(* PLC project Unnamed, Unknown Unnamed 1 *)
(* stored: creationDateTime 2025-11-17T12:43:33, modificationDateTime 2025-11-17T18:21:39 *)

PROGRAM Lab1
  VAR
    btn AT %IX0.0 : BOOL := False;
  END_VAR
  VAR
    AllowedPress : BOOL := False;
    pressed : BOOL := False;
    Ped_wait : BOOL := False;
    Pedestrian : BOOL := False;
  END_VAR
  VAR
    north AT %QX0.0 : BOOL := False;
    south AT %QX0.1 : BOOL := False;
    west AT %QX0.2 : BOOL := False;
    east AT %QX0.3 : BOOL := False;
  END_VAR
  VAR
    state : BOOL := False;
    S0 : BOOL := False;
    S1 : BOOL := False;
    T10 : TIME := T#10s;
    T80 : TIME := T#80s;
    Allowed_timer : BOOL := False;
    Timer_cooldown : BOOL := False;
    FF1 : BOOL := False;
    FF2 : BOOL := False;
    FF_output : BOOL := False;
    TON0 : TON;
    TON1 : TON;
    TP0 : TP;
    TP1 : TP;
    R_TRIG1 : R_TRIG;
    R_TRIG0 : R_TRIG;
    R_TRIG2 : R_TRIG;
    R_TRIG3 : R_TRIG;
    R_TRIG4 : R_TRIG;
    R_TRIG5 : R_TRIG;
  END_VAR

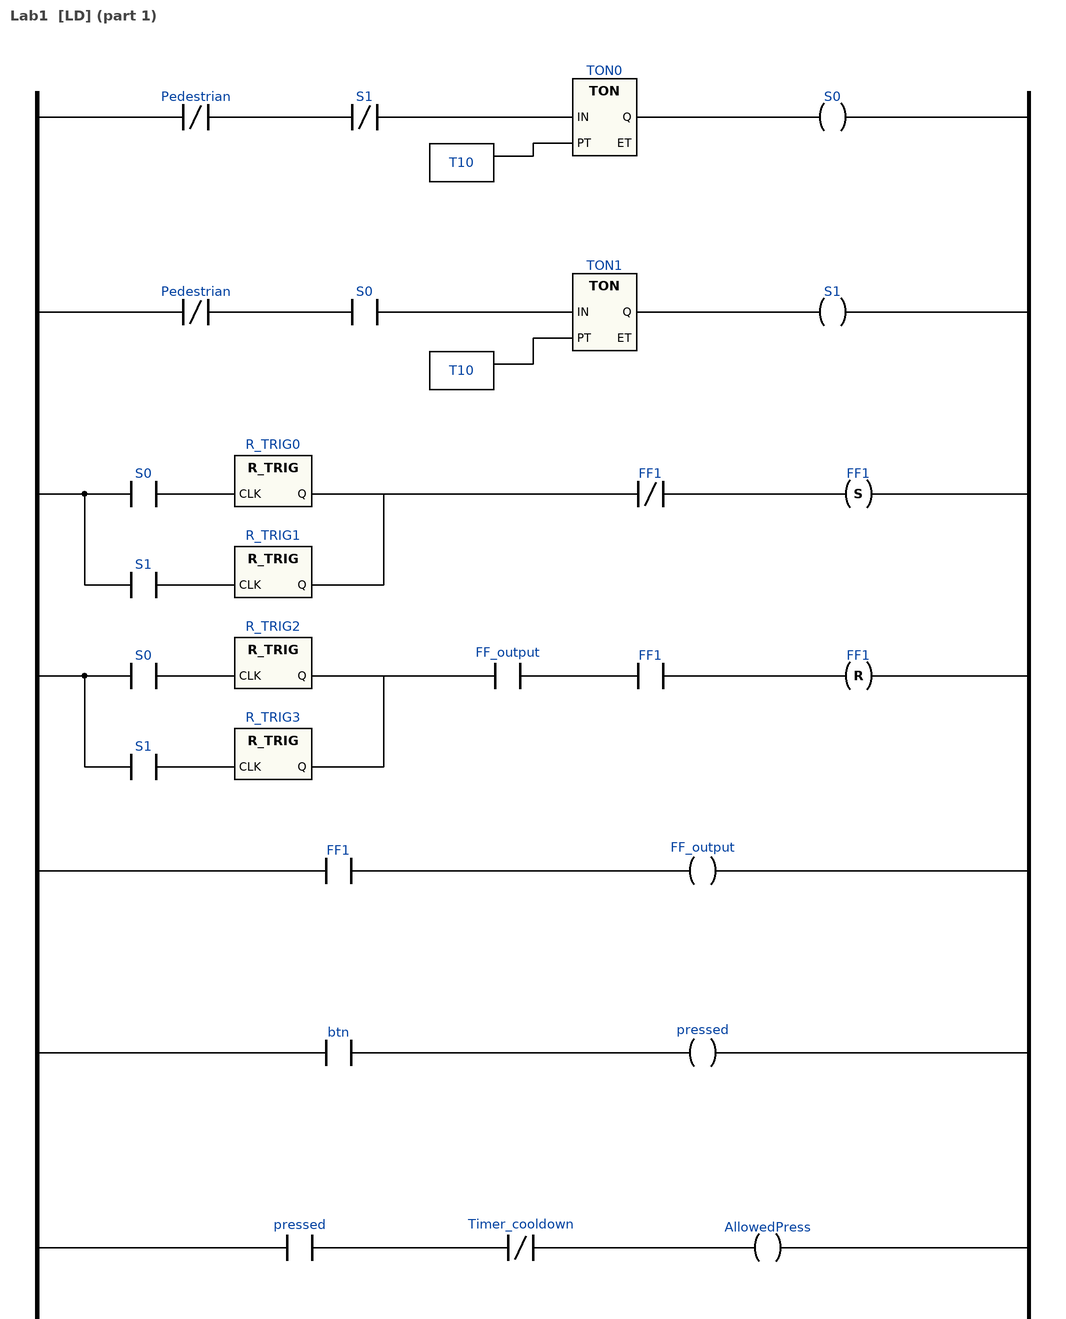
(* LD diagram, written out as Structured Text *)
TON0(IN := NOT Pedestrian AND NOT S1, PT := T10);
S0 := TON0.Q;
TON1(IN := NOT Pedestrian AND S0, PT := T10);
S1 := TON1.Q;
R_TRIG1(CLK := S1);
R_TRIG0(CLK := S0);
IF (R_TRIG1.Q OR R_TRIG0.Q) AND NOT FF1 THEN FF1 := TRUE; END_IF;
R_TRIG2(CLK := S0);
R_TRIG3(CLK := S1);
IF (R_TRIG2.Q OR R_TRIG3.Q) AND FF_output AND FF1 THEN FF1 := FALSE; END_IF;
FF_output := FF1;
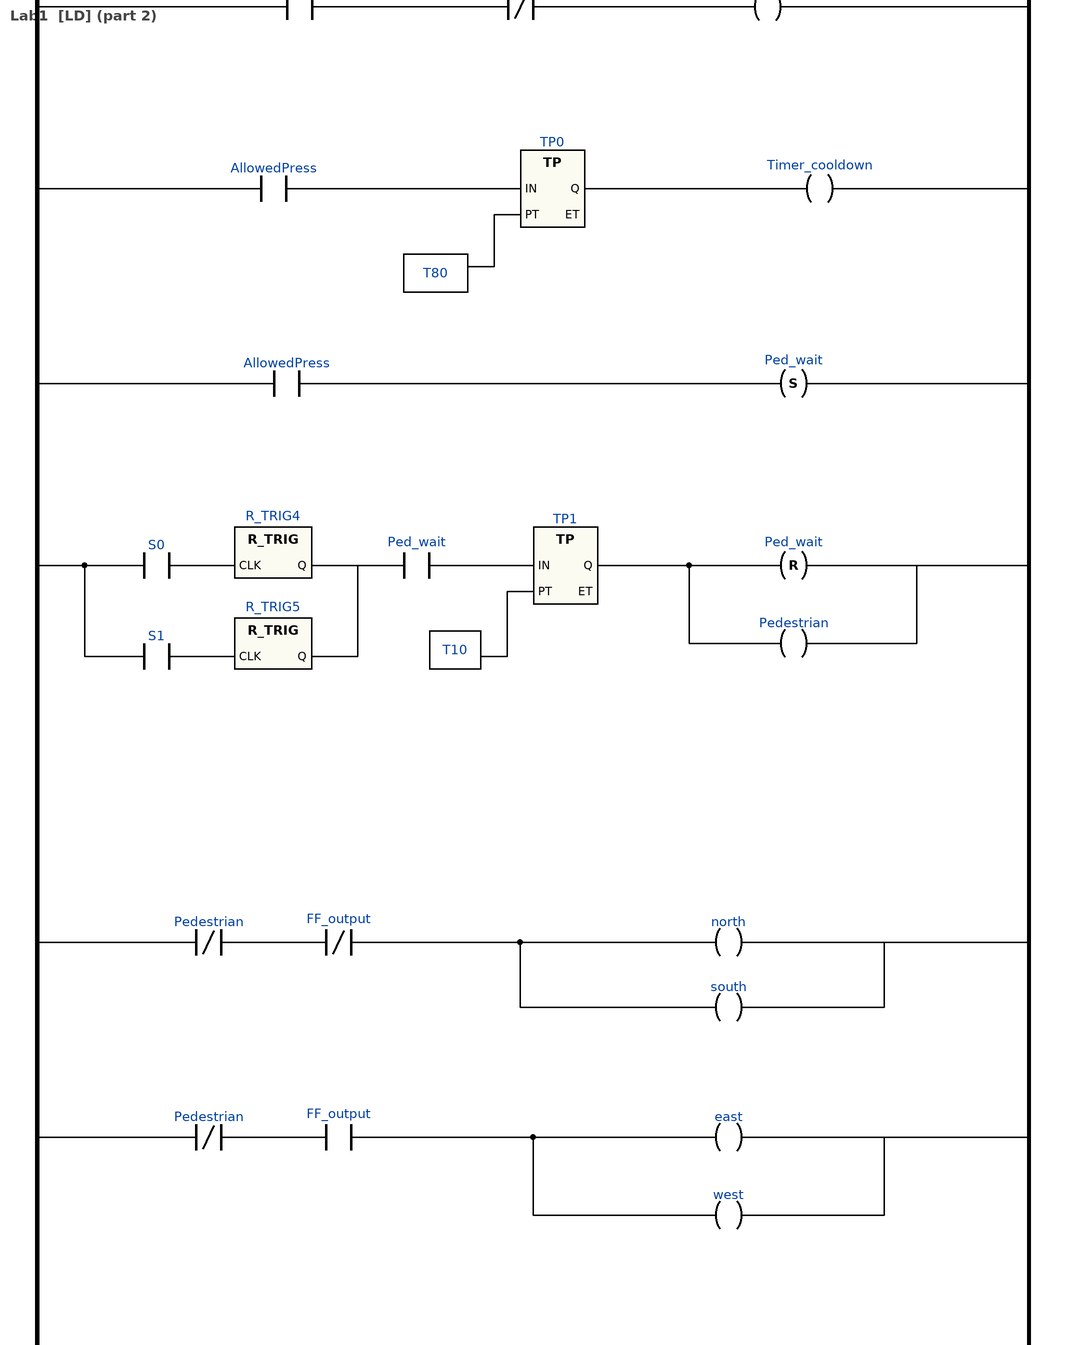
north := NOT Pedestrian AND NOT FF_output;
south := NOT Pedestrian AND NOT FF_output;
east := NOT Pedestrian AND FF_output;
west := NOT Pedestrian AND FF_output;
pressed := btn;
AllowedPress := pressed AND NOT Timer_cooldown;
TP0(IN := AllowedPress, PT := T80);
Timer_cooldown := TP0.Q;
IF AllowedPress THEN Ped_wait := TRUE; END_IF;
R_TRIG5(CLK := S1);
R_TRIG4(CLK := S0);
TP1(IN := (R_TRIG5.Q OR R_TRIG4.Q) AND Ped_wait, PT := T10);
IF TP1.Q THEN Ped_wait := FALSE; END_IF;
Pedestrian := TP1.Q;
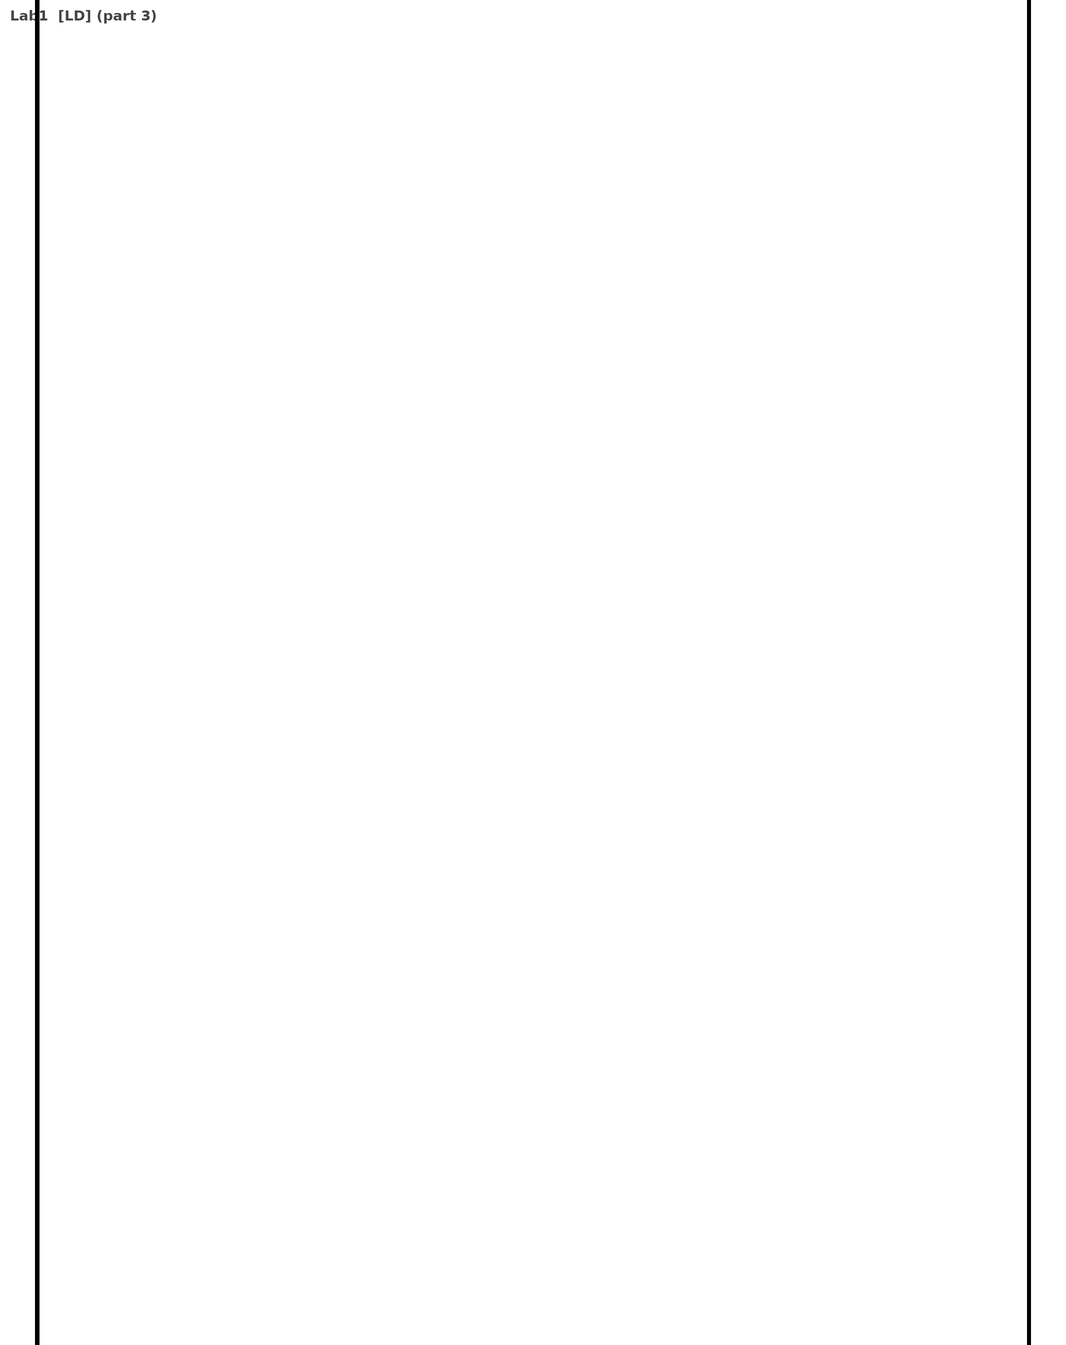
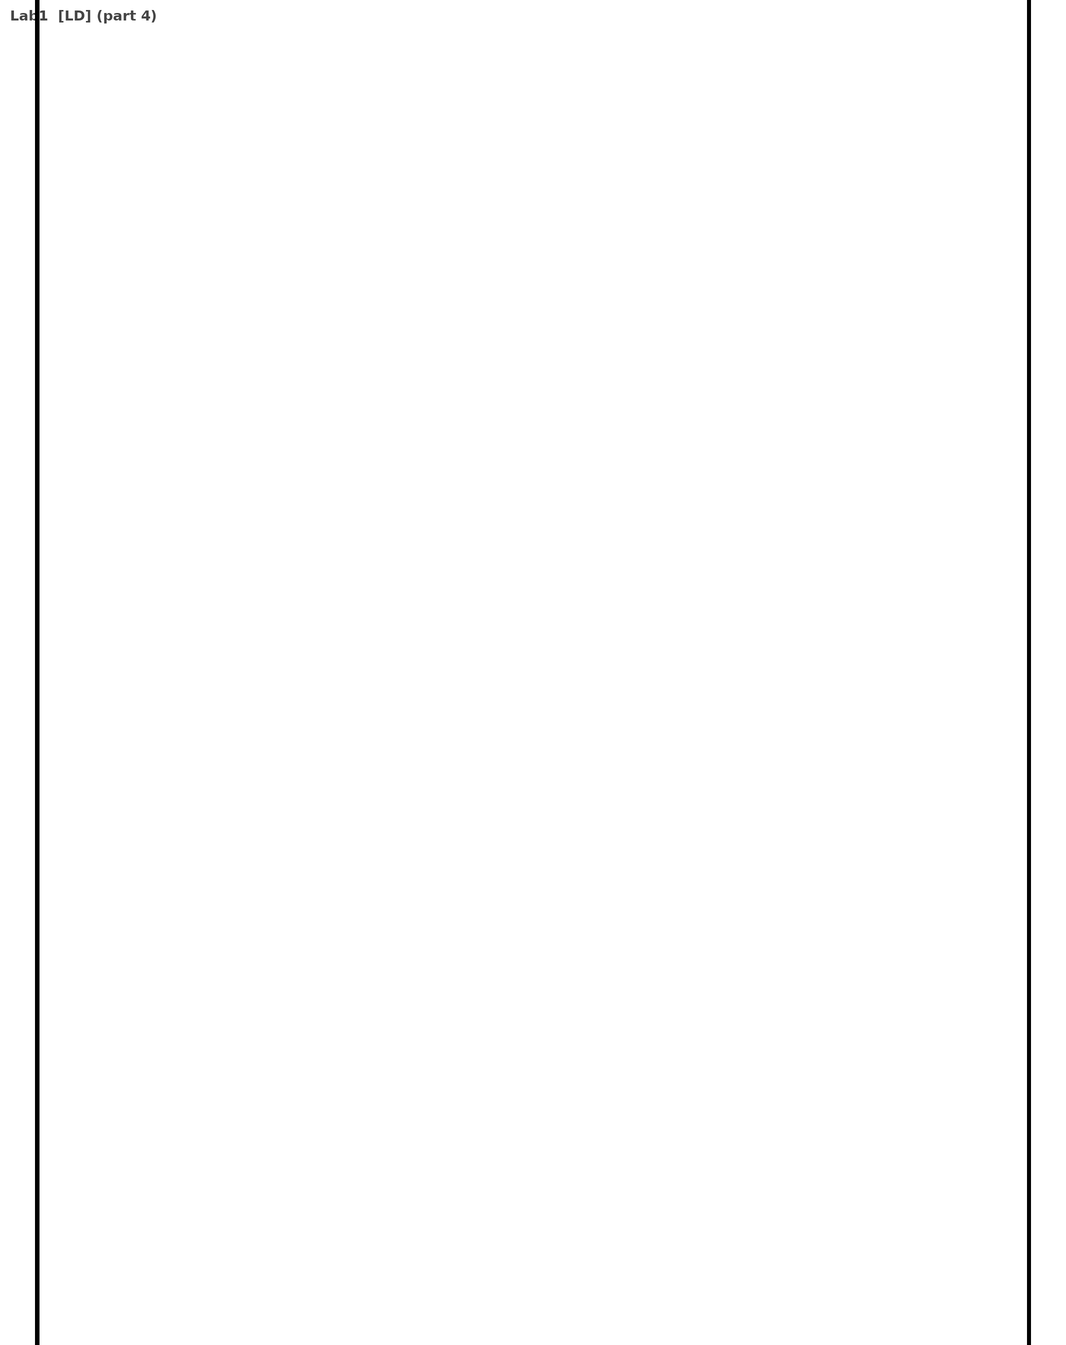
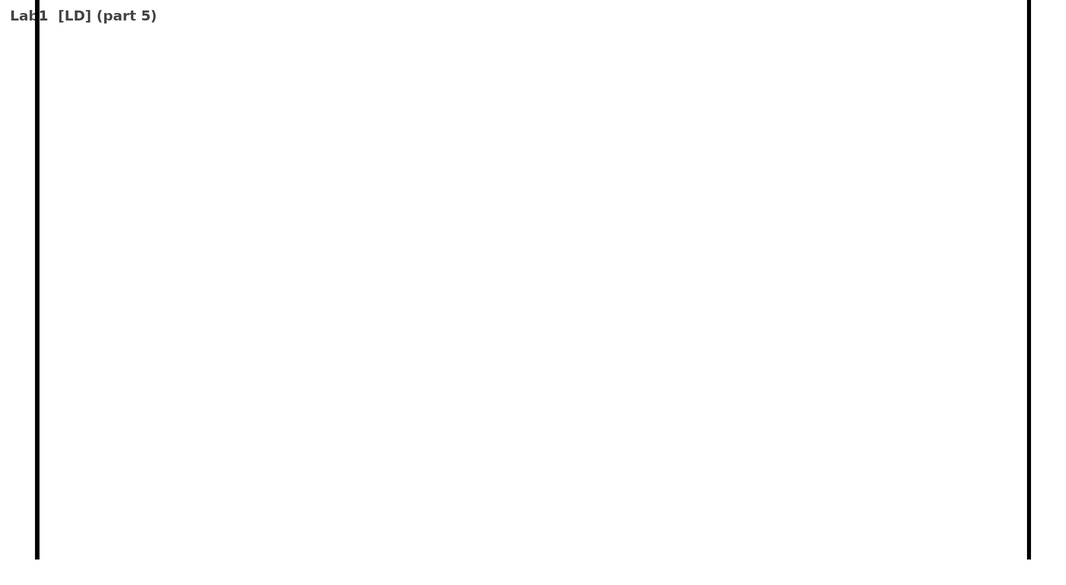
END_PROGRAM

CONFIGURATION Config0
  RESOURCE Res0 ON PLC
    TASK task0(INTERVAL := T#20ms, PRIORITY := 0);
    PROGRAM instance0 WITH task0 : Lab1;
  END_RESOURCE
END_CONFIGURATION
